// TIA Portal V16 export
// export: Created 2022-11-17T15:49:12.4725311Z, ExportSetting WithDefaults, DisplayName Totally Integrated Automation Portal, DisplayVersion V16 Update 6, DisplayName TIA Portal Version Control Interface, DisplayVersion V16 Update 2, DisplayName TIA Portal Openness, DisplayVersion V16 Update 6, DisplayName SINAMICS Startdrive Advanced, DisplayVersion V16 Update 5, DisplayName SINAMICS Startdrive G130, G150, S120, S150, SINAMICS MV, S210, DisplayVersion V16 Update 5, DisplayName SINAMICS Startdrive G110M, G120, G120C, G120D, G120P, G115D, DisplayVersion V16 Update 5, DisplayName STEP 7 Professional, DisplayVersion V16 Update 6, DisplayName STEP 7 Safety, DisplayVersion V16, DisplayName WinCC Advanced, DisplayVersion V16 Update 6
FUNCTION "FC02_Technoplat_TandC" : Void   // FC2, LAD
TITLE = Technoplat timer and counter
{ S7_Optimized_Access := 'FALSE' }
AUTHOR : Robopac
VERSION : 0.0
// stored: AutoNumber false, IsIECCheckEnabled false, SetENOAutomatically false, UDAEnableTagReadback false
   VAR_INPUT
      FASTSPEED : Bool;
   END_VAR
   VAR_TEMP
      TempInt : Int;
      TempDint : DInt;
   END_VAR
   VAR_TEMP   // added for the SCL form of the ladder/FBD networks
      _w1 : Bool;
      _w2 : Bool;
   END_VAR
BEGIN

REGION Network 1: Time to filter inverter alarms
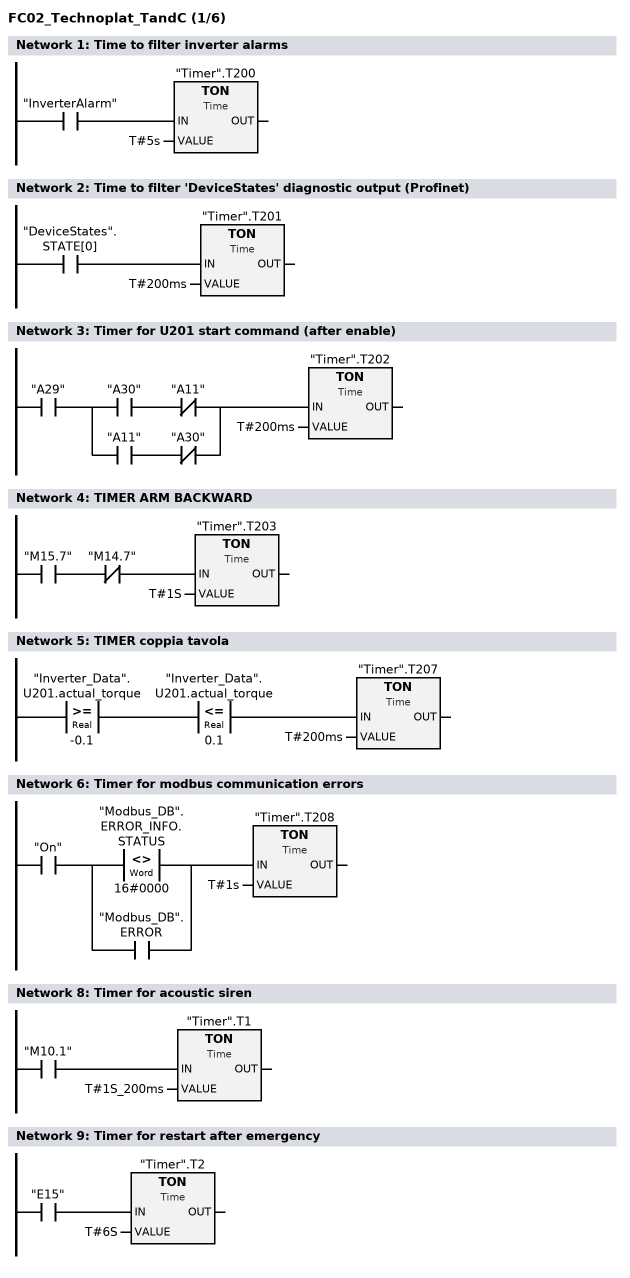
   "Timer".T200.TON(IN := "InverterAlarm", PT := T#5s);   // TON coil
END_REGION

REGION Network 2: Time to filter 'DeviceStates' diagnostic output (Profinet)
   "Timer".T201.TON(IN := "DeviceStates".STATE[0], PT := T#200ms);   // TON coil
END_REGION

REGION Network 3: Timer for U201 start command (after enable)
   "Timer".T202.TON(IN := "A29" AND (("A30" AND NOT "A11") OR ("A11" AND NOT "A30")), PT := T#200ms);   // TON coil
END_REGION

REGION Network 4: TIMER ARM BACKWARD
   "Timer".T203.TON(IN := "M15.7" AND NOT "M14.7", PT := T#1S);   // TON coil
END_REGION

REGION Network 5: TIMER coppia tavola
   "Timer".T207.TON(IN := ("Inverter_Data".U201.actual_torque >= (-0.1)) AND ("Inverter_Data".U201.actual_torque <= 0.1), PT := T#200ms);   // TON coil
END_REGION

REGION Network 6: Timer for modbus communication errors
   "Timer".T208.TON(IN := "On" AND (("Modbus_DB".ERROR_INFO.STATUS <> 16#0000) OR "Modbus_DB".ERROR), PT := T#1s);   // TON coil
END_REGION

REGION Network 7: TECHNOPLAT3000
END_REGION

REGION Network 8: Timer for acoustic siren
   "Timer".T1.TON(IN := "M10.1", PT := T#1S_200ms);   // TON coil
END_REGION

REGION Network 9: Timer for restart after emergency
   "Timer".T2.TON(IN := "E15", PT := T#6S);   // TON coil
END_REGION

REGION Network 10: Timer to reset emergency
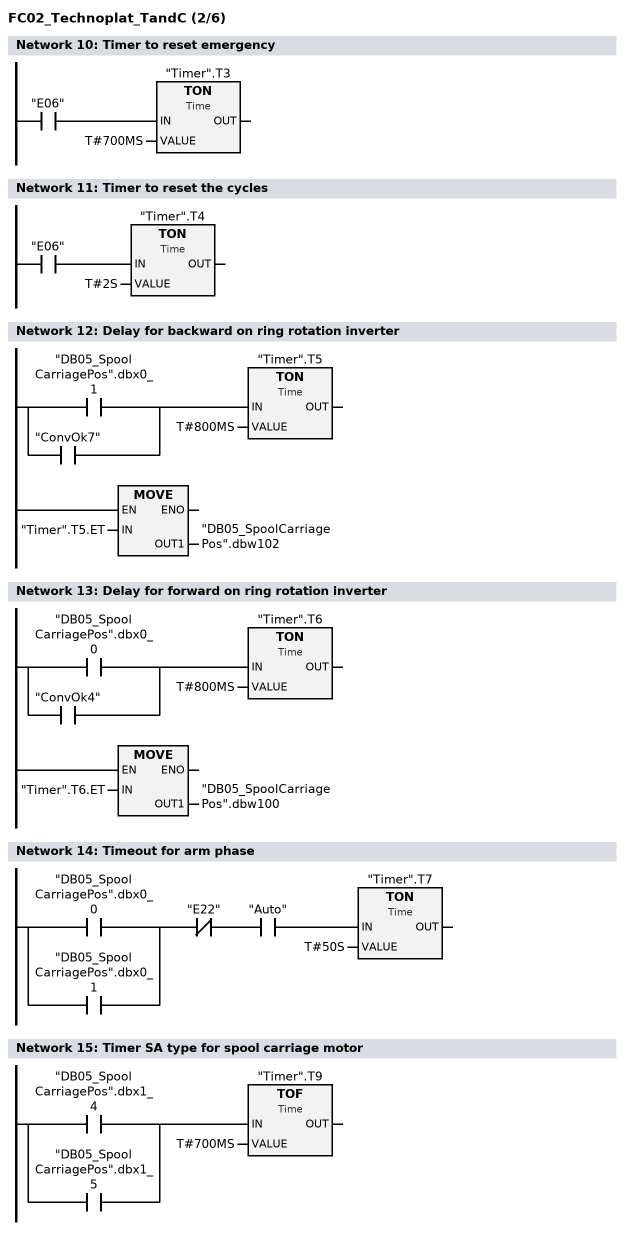
   "Timer".T3.TON(IN := "E06", PT := T#700MS);   // TON coil
END_REGION

REGION Network 11: Timer to reset the cycles
   "Timer".T4.TON(IN := "E06", PT := T#2S);   // TON coil
END_REGION

REGION Network 12: Delay for backward on ring rotation inverter
   "Timer".T5.TON(IN := "DB05_SpoolCarriagePos".dbx0_1 OR "ConvOk7", PT := T#800MS);   // TON coil
   "DB05_SpoolCarriagePos".dbw102 := "Timer".T5.ET;
END_REGION

REGION Network 13: Delay for forward on ring rotation inverter
   "Timer".T6.TON(IN := "DB05_SpoolCarriagePos".dbx0_0 OR "ConvOk4", PT := T#800MS);   // TON coil
   "DB05_SpoolCarriagePos".dbw100 := "Timer".T6.ET;
END_REGION

REGION Network 14: Timeout for arm phase
   "Timer".T7.TON(IN := ("DB05_SpoolCarriagePos".dbx0_0 OR "DB05_SpoolCarriagePos".dbx0_1) AND NOT "E22" AND "Auto", PT := T#50S);   // TON coil
END_REGION

REGION Network 15: Timer SA type for spool carriage motor
   "Timer".T9.TOF(IN := "DB05_SpoolCarriagePos".dbx1_4 OR "DB05_SpoolCarriagePos".dbx1_5, PT := T#700MS);   // TOF coil
END_REGION

REGION Network 16: Timer SA type for arm rotation motor
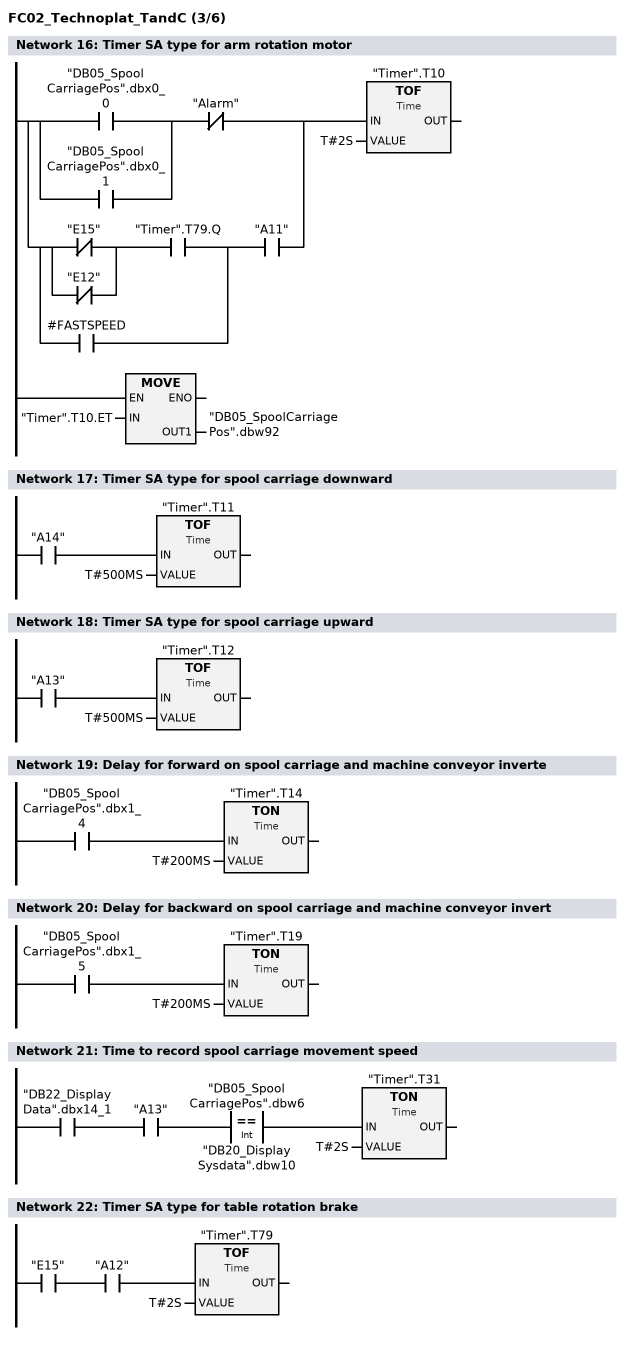
   "Timer".T10.TOF(IN := (("DB05_SpoolCarriagePos".dbx0_0 OR "DB05_SpoolCarriagePos".dbx0_1) AND NOT "Alarm") OR ((((NOT "E15" OR NOT "E12") AND "Timer".T79.Q) OR #FASTSPEED) AND "A11"), PT := T#2S);   // TOF coil
   "DB05_SpoolCarriagePos".dbw92 := "Timer".T10.ET;
END_REGION

REGION Network 17: Timer SA type for spool carriage downward
   "Timer".T11.TOF(IN := "A14", PT := T#500MS);   // TOF coil
END_REGION

REGION Network 18: Timer SA type for spool carriage upward
   "Timer".T12.TOF(IN := "A13", PT := T#500MS);   // TOF coil
END_REGION

REGION Network 19: Delay for forward on spool carriage and machine conveyor inverte
   "Timer".T14.TON(IN := "DB05_SpoolCarriagePos".dbx1_4, PT := T#200MS);   // TON coil
END_REGION

REGION Network 20: Delay for backward on spool carriage and machine conveyor invert
   "Timer".T19.TON(IN := "DB05_SpoolCarriagePos".dbx1_5, PT := T#200MS);   // TON coil
END_REGION

REGION Network 21: Time to record spool carriage movement speed
   "Timer".T31.TON(IN := "DB22_DisplayData".dbx14_1 AND "A13" AND ("DB05_SpoolCarriagePos".dbw6 = "DB20_DisplaySysdata".dbw10), PT := T#2S);   // TON coil
END_REGION

REGION Network 22: Timer SA type for table rotation brake
   "Timer".T79.TOF(IN := "E15" AND "A12", PT := T#2S);   // TOF coil
END_REGION

REGION Network 23: T87: Timer for slow conveyor manual movement
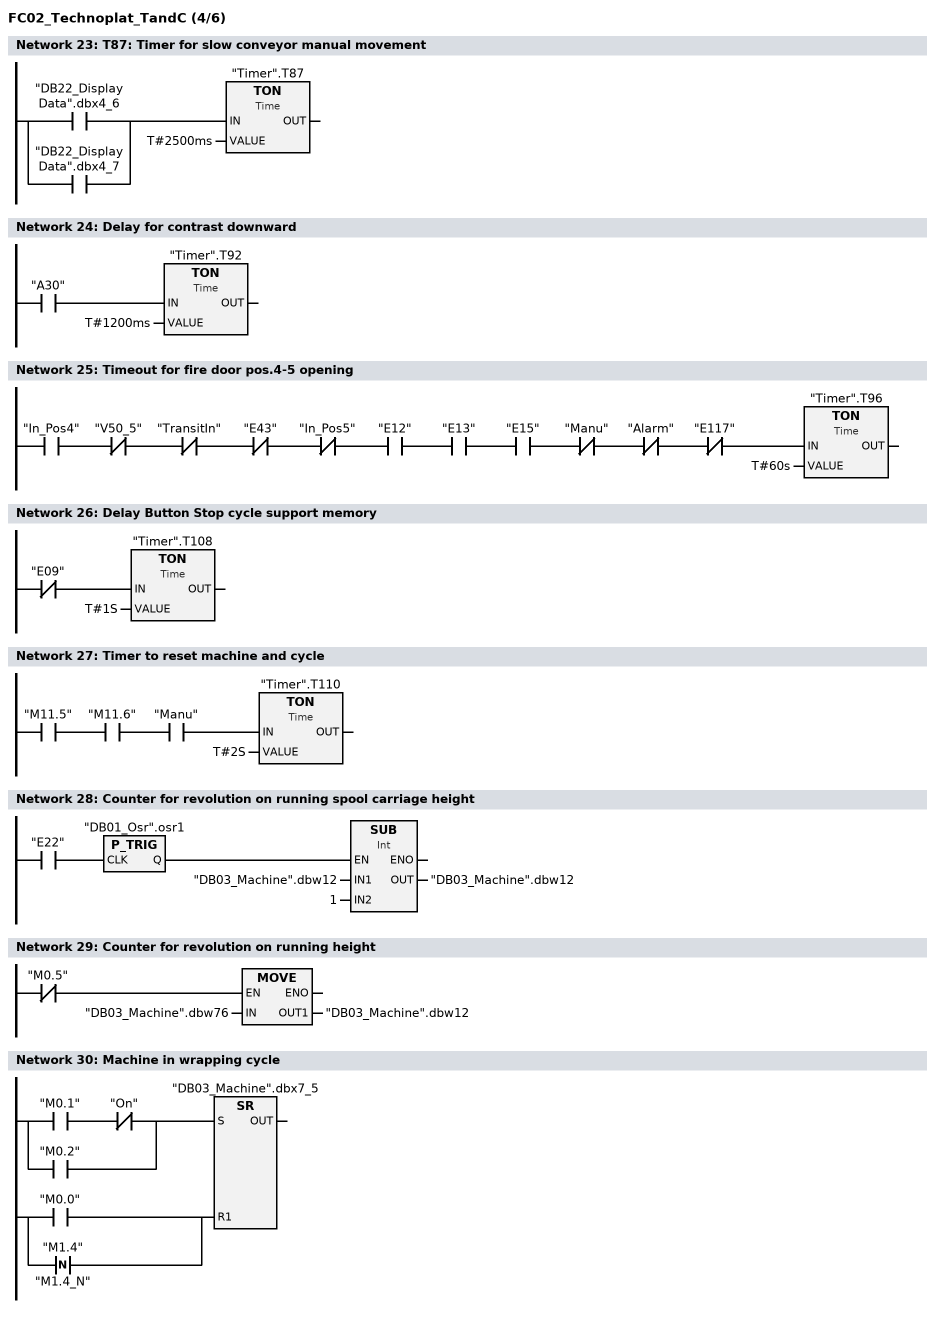
   "Timer".T87.TON(IN := "DB22_DisplayData".dbx4_6 OR "DB22_DisplayData".dbx4_7, PT := T#2500ms);   // TON coil
END_REGION

REGION Network 24: Delay for contrast downward
   "Timer".T92.TON(IN := "A30", PT := T#1200ms);   // TON coil
END_REGION

REGION Network 25: Timeout for fire door pos.4-5 opening
   "Timer".T96.TON(IN := "In_Pos4" AND NOT "V50_5" AND NOT "TransitIn" AND NOT "E43" AND NOT "In_Pos5" AND "E12" AND "E13" AND "E15" AND NOT "Manu" AND NOT "Alarm" AND NOT "E117", PT := T#60s);   // TON coil
END_REGION

REGION Network 26: Delay Button Stop cycle support memory
   "Timer".T108.TON(IN := NOT "E09", PT := T#1S);   // TON coil
END_REGION

REGION Network 27: Timer to reset machine and cycle
   "Timer".T110.TON(IN := "M11.5" AND "M11.6" AND "Manu", PT := T#2S);   // TON coil
END_REGION

REGION Network 28: Counter for revolution on running spool carriage height
   RUNG wire#powerrail
      Contact( "E22" )
      P_Trig( "DB01_Osr".osr1 )
      { S7_Templates := "SrcType := Int"; S7_GenerateENO := "TRUE" } Sub(in1 := "DB03_Machine".dbw12, in2 := 1, out => "DB03_Machine".dbw12)
   END_RUNG
   // the same network as SCL:
   #_w1 := "E22" AND NOT "DB01_Osr".osr1;   // rising edge
   "DB01_Osr".osr1 := "E22";
   IF #_w1 THEN "DB03_Machine".dbw12 := "DB03_Machine".dbw12 - 1; END_IF;
END_REGION

REGION Network 29: Counter for revolution on running height
   RUNG wire#powerrail
      I_Contact( "M0.5" )
      { S7_GenerateENO := "TRUE" } Move(in := "DB03_Machine".dbw76, out1 => "DB03_Machine".dbw12)
   END_RUNG
   // the same network as SCL:
   IF NOT "M0.5" THEN "DB03_Machine".dbw12 := "DB03_Machine".dbw76; END_IF;
END_REGION

REGION Network 30: Machine in wrapping cycle
   RUNG wire#powerrail
      Contact( "M0.1" )
      I_Contact( "On" )
      wire#w1
      S_SR(operand := "DB03_Machine".dbx7_5, r1 := wire#w2)
   END_RUNG
   RUNG wire#powerrail
      Contact( "M0.2" )
   END_RUNG wire#w1
   RUNG wire#powerrail
      Contact( "M0.0" )
   END_RUNG wire#w2
   RUNG wire#powerrail
      N_Contact(operand := "M1.4", bit := "M1.4_N")
   END_RUNG wire#w2
   // the same network as SCL:
   #_w1 := NOT "M1.4" AND "M1.4_N";   // falling edge of "M1.4"
   "M1.4_N" := "M1.4";
   IF ("M0.1" AND NOT "On") OR "M0.2" THEN
       "DB03_Machine".dbx7_5 := TRUE;   // SR flip-flop
   END_IF;
   IF "M0.0" OR #_w1 THEN "DB03_Machine".dbx7_5 := FALSE; END_IF;
END_REGION

REGION Network 31: Support memory to refresh pallet per hour value
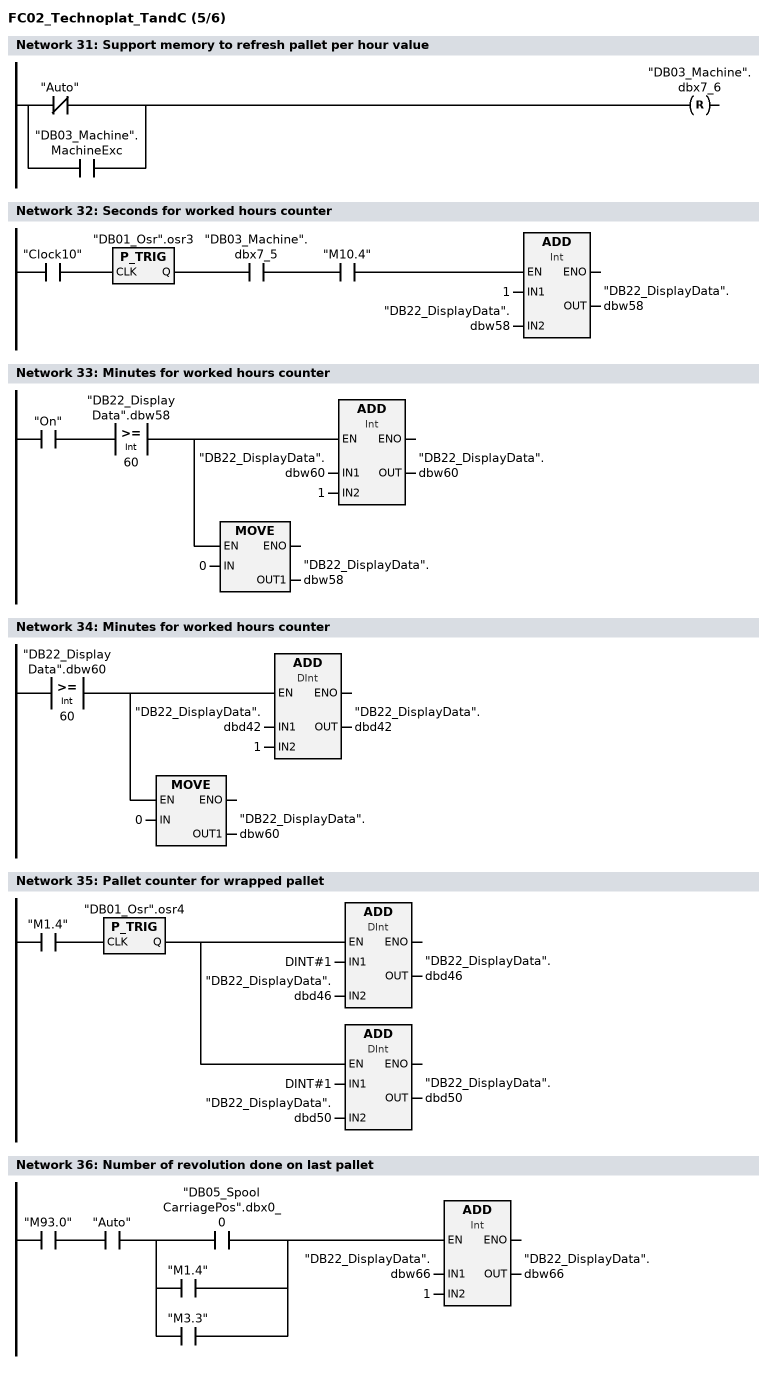
   RUNG wire#powerrail
      I_Contact( "Auto" )
      wire#w1
      R_Coil( "DB03_Machine".dbx7_6 )
   END_RUNG
   RUNG wire#powerrail
      Contact( "DB03_Machine".MachineExc )
   END_RUNG wire#w1
   // the same network as SCL:
   IF NOT "Auto" OR "DB03_Machine".MachineExc THEN "DB03_Machine".dbx7_6 := FALSE; END_IF;
END_REGION

REGION Network 32: Seconds for worked hours counter
   RUNG wire#powerrail
      Contact( "Clock10" )
      P_Trig( "DB01_Osr".osr3 )
      Contact( "DB03_Machine".dbx7_5 )
      Contact( "M10.4" )
      { S7_Templates := "SrcType := Int"; S7_GenerateENO := "TRUE" } Add(in1 := 1, in2 := "DB22_DisplayData".dbw58, out => "DB22_DisplayData".dbw58)
   END_RUNG
   // the same network as SCL:
   #_w1 := "Clock10" AND NOT "DB01_Osr".osr3;   // rising edge
   "DB01_Osr".osr3 := "Clock10";
   IF #_w1 AND "DB03_Machine".dbx7_5 AND "M10.4" THEN
       "DB22_DisplayData".dbw58 := 1 + "DB22_DisplayData".dbw58;
   END_IF;
END_REGION

REGION Network 33: Minutes for worked hours counter
   RUNG wire#powerrail
      Contact( "On" )
      { S7_Templates := "SrcType := Int" } GE_Contact(in1 := "DB22_DisplayData".dbw58, in2 := 60)
      wire#w1
      { S7_Templates := "SrcType := Int"; S7_GenerateENO := "TRUE" } Add(in1 := "DB22_DisplayData".dbw60, in2 := 1, out => "DB22_DisplayData".dbw60)
   END_RUNG
   RUNG wire#w1
      { S7_GenerateENO := "TRUE" } Move(in := 0, out1 => "DB22_DisplayData".dbw58)
   END_RUNG
   // the same network as SCL:
   IF "On" AND ("DB22_DisplayData".dbw58 >= 60) THEN
       "DB22_DisplayData".dbw60 := "DB22_DisplayData".dbw60 + 1;
       "DB22_DisplayData".dbw58 := 0;
   END_IF;
END_REGION

REGION Network 34: Minutes for worked hours counter
   RUNG wire#powerrail
      { S7_Templates := "SrcType := Int" } GE_Contact(in1 := "DB22_DisplayData".dbw60, in2 := 60)
      wire#w1
      { S7_Templates := "SrcType := DInt"; S7_GenerateENO := "TRUE" } Add(in1 := "DB22_DisplayData".dbd42, in2 := 1, out => "DB22_DisplayData".dbd42)
   END_RUNG
   RUNG wire#w1
      { S7_GenerateENO := "TRUE" } Move(in := 0, out1 => "DB22_DisplayData".dbw60)
   END_RUNG
   // the same network as SCL:
   IF "DB22_DisplayData".dbw60 >= 60 THEN
       "DB22_DisplayData".dbd42 := "DB22_DisplayData".dbd42 + 1;
       "DB22_DisplayData".dbw60 := 0;
   END_IF;
END_REGION

REGION Network 35: Pallet counter for wrapped pallet
   RUNG wire#powerrail
      Contact( "M1.4" )
      P_Trig( "DB01_Osr".osr4 )
      wire#w1
      { S7_Templates := "SrcType := DInt"; S7_GenerateENO := "TRUE" } Add(in1 := DINT#1, in2 := "DB22_DisplayData".dbd46, out => "DB22_DisplayData".dbd46)
   END_RUNG
   RUNG wire#w1
      { S7_Templates := "SrcType := DInt"; S7_GenerateENO := "TRUE" } Add(in1 := DINT#1, in2 := "DB22_DisplayData".dbd50, out => "DB22_DisplayData".dbd50)
   END_RUNG
   // the same network as SCL:
   #_w1 := "M1.4" AND NOT "DB01_Osr".osr4;   // rising edge
   "DB01_Osr".osr4 := "M1.4";
   IF #_w1 THEN
       "DB22_DisplayData".dbd46 := DINT#1 + "DB22_DisplayData".dbd46;
       "DB22_DisplayData".dbd50 := DINT#1 + "DB22_DisplayData".dbd50;
   END_IF;
END_REGION

REGION Network 36: Number of revolution done on last pallet
   RUNG wire#powerrail
      Contact( "M93.0" )
      Contact( "Auto" )
      wire#w1
      Contact( "DB05_SpoolCarriagePos".dbx0_0 )
      wire#w2
      { S7_Templates := "SrcType := Int"; S7_GenerateENO := "TRUE" } Add(in1 := "DB22_DisplayData".dbw66, in2 := 1, out => "DB22_DisplayData".dbw66)
   END_RUNG
   RUNG wire#w1
      Contact( "M1.4" )
   END_RUNG wire#w2
   RUNG wire#w1
      Contact( "M3.3" )
   END_RUNG wire#w2
   // the same network as SCL:
   IF "M93.0" AND "Auto" AND ("DB05_SpoolCarriagePos".dbx0_0 OR "M1.4" OR "M3.3") THEN
       "DB22_DisplayData".dbw66 := "DB22_DisplayData".dbw66 + 1;
   END_IF;
END_REGION

REGION Network 37: Number of revolution done on last pallet
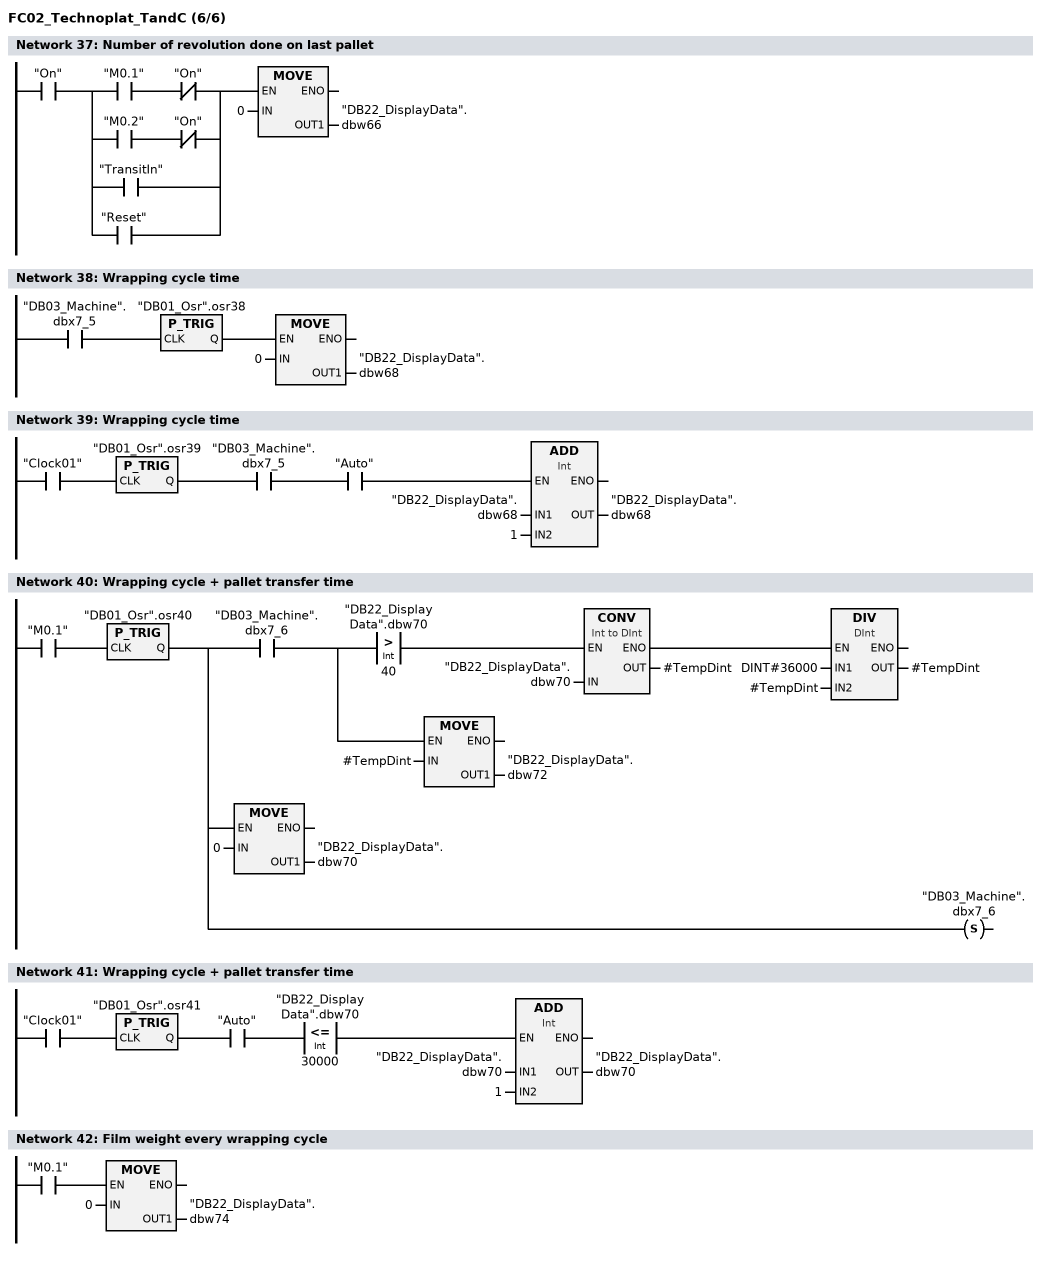
   RUNG wire#powerrail
      Contact( "On" )
      wire#w1
      Contact( "M0.1" )
      I_Contact( "On" )
      wire#w2
      { S7_GenerateENO := "TRUE" } Move(in := 0, out1 => "DB22_DisplayData".dbw66)
   END_RUNG
   RUNG wire#w1
      Contact( "M0.2" )
      I_Contact( "On" )
   END_RUNG wire#w2
   RUNG wire#w1
      Contact( "TransitIn" )
   END_RUNG wire#w2
   RUNG wire#w1
      Contact( "Reset" )
   END_RUNG wire#w2
   // the same network as SCL:
   IF "On" AND (("M0.1" AND NOT "On") OR ("M0.2" AND NOT "On") OR "TransitIn" OR "Reset") THEN
       "DB22_DisplayData".dbw66 := 0;
   END_IF;
END_REGION

REGION Network 38: Wrapping cycle time
   RUNG wire#powerrail
      Contact( "DB03_Machine".dbx7_5 )
      P_Trig( "DB01_Osr".osr38 )
      { S7_GenerateENO := "TRUE" } Move(in := 0, out1 => "DB22_DisplayData".dbw68)
   END_RUNG
   // the same network as SCL:
   #_w1 := "DB03_Machine".dbx7_5 AND NOT "DB01_Osr".osr38;   // rising edge
   "DB01_Osr".osr38 := "DB03_Machine".dbx7_5;
   IF #_w1 THEN "DB22_DisplayData".dbw68 := 0; END_IF;
END_REGION

REGION Network 39: Wrapping cycle time
   RUNG wire#powerrail
      Contact( "Clock01" )
      P_Trig( "DB01_Osr".osr39 )
      Contact( "DB03_Machine".dbx7_5 )
      Contact( "Auto" )
      { S7_Templates := "SrcType := Int"; S7_GenerateENO := "TRUE" } Add(in1 := "DB22_DisplayData".dbw68, in2 := 1, out => "DB22_DisplayData".dbw68)
   END_RUNG
   // the same network as SCL:
   #_w1 := "Clock01" AND NOT "DB01_Osr".osr39;   // rising edge
   "DB01_Osr".osr39 := "Clock01";
   IF #_w1 AND "DB03_Machine".dbx7_5 AND "Auto" THEN
       "DB22_DisplayData".dbw68 := "DB22_DisplayData".dbw68 + 1;
   END_IF;
END_REGION

REGION Network 40: Wrapping cycle + pallet transfer time
   RUNG wire#powerrail
      Contact( "M0.1" )
      P_Trig( "DB01_Osr".osr40 )
      wire#w1
      Contact( "DB03_Machine".dbx7_6 )
      wire#w2
      { S7_Templates := "SrcType := Int" } GT_Contact(in1 := "DB22_DisplayData".dbw70, in2 := 40)
      { S7_Templates := "[SrcType := Int, DestType := DInt]"; S7_GenerateENO := "TRUE" } Convert(in := "DB22_DisplayData".dbw70, out => #TempDint)
      { S7_Templates := "SrcType := DInt"; S7_GenerateENO := "TRUE" } Div(in1 := DINT#36000, in2 := #TempDint, out => #TempDint)
   END_RUNG
   RUNG wire#w2
      { S7_GenerateENO := "TRUE" } Move(in := #TempDint, out1 => "DB22_DisplayData".dbw72)
   END_RUNG
   RUNG wire#w1
      { S7_GenerateENO := "TRUE" } Move(in := 0, out1 => "DB22_DisplayData".dbw70)
   END_RUNG
   RUNG wire#w1
      S_Coil( "DB03_Machine".dbx7_6 )
   END_RUNG
   // the same network as SCL:
   // ENO of a box is taken as its EN; it also drops when the box reports an error
   #_w1 := "M0.1" AND NOT "DB01_Osr".osr40;   // rising edge
   "DB01_Osr".osr40 := "M0.1";
   #_w2 := #_w1 AND "DB03_Machine".dbx7_6;
   IF #_w2 AND ("DB22_DisplayData".dbw70 > 40) THEN
       #TempDint := INT_TO_DINT("DB22_DisplayData".dbw70);
       #TempDint := DINT#36000 / #TempDint;
   END_IF;
   IF #_w2 THEN "DB22_DisplayData".dbw72 := #TempDint; END_IF;
   IF #_w1 THEN
       "DB22_DisplayData".dbw70 := 0;
       "DB03_Machine".dbx7_6 := TRUE;
   END_IF;
END_REGION

REGION Network 41: Wrapping cycle + pallet transfer time
   RUNG wire#powerrail
      Contact( "Clock01" )
      P_Trig( "DB01_Osr".osr41 )
      Contact( "Auto" )
      { S7_Templates := "SrcType := Int" } LE_Contact(in1 := "DB22_DisplayData".dbw70, in2 := 30000)
      { S7_Templates := "SrcType := Int"; S7_GenerateENO := "TRUE" } Add(in1 := "DB22_DisplayData".dbw70, in2 := 1, out => "DB22_DisplayData".dbw70)
   END_RUNG
   // the same network as SCL:
   #_w1 := "Clock01" AND NOT "DB01_Osr".osr41;   // rising edge
   "DB01_Osr".osr41 := "Clock01";
   IF #_w1 AND "Auto" AND ("DB22_DisplayData".dbw70 <= 30000) THEN
       "DB22_DisplayData".dbw70 := "DB22_DisplayData".dbw70 + 1;
   END_IF;
END_REGION

REGION Network 42: Film weight every wrapping cycle
   RUNG wire#powerrail
      Contact( "M0.1" )
      { S7_GenerateENO := "TRUE" } Move(in := 0, out1 => "DB22_DisplayData".dbw74)
   END_RUNG
   // the same network as SCL:
   IF "M0.1" THEN "DB22_DisplayData".dbw74 := 0; END_IF;
END_REGION
END_FUNCTION
